(*
	dont we all?
*)
INTERFACE IHaveUlintValue EXTENDS CNM_AbstractObject.IObject

PROPERTY value : ULINT
GET
END_GET
SET
END_SET
END_PROPERTY

END_INTERFACE

(* stored: Version 1.1.0.1
   Itf IHaveUlintValue: Id {f705222f-5fce-45b1-95d7-5ab59ce05c6f}
   Property value: Id {cf46b51f-37c0-4bba-a4cf-97f579adb3c7}
   Get Get: Id {162cab22-fbd3-4f4d-91e2-77fa925b13b0}
   Set Set: Id {12510490-aa8c-416e-a741-05448fc97d25} *)
